{attribute addProperty BoxType "EPP3314-0002-0016"}
{attribute addProperty Id "TC_Inputs_ChannelAT %I*ARRAY[0..6] OF TC_Inputs_Channel_F16A160D128160WcStateAT %I*WcState_98A4DF7520.250InfoDataAT %I*InfoData_BC63D37F80100"}
{attribute addProperty CRC "2970462671"}
{attribute addProperty SizeInBites "210"}
{attribute addProperty SizeInBytes "26.25"}
TYPE EPP3314_A69716D7 :
STRUCT
	{attribute addProperty Name "TC_Inputs_Channel"}
	TC_Inputs_Channel : ARRAY[0..6] OF TC_Inputs_Channel_F16A160D;
	{attribute addProperty Name "WcState"}
	WcState : WcState_98A4DF75;
	{attribute addProperty Name "InfoData"}
	InfoData : InfoData_BC63D37F;
END_STRUCT
END_TYPE

(* stored: Version 1.2.0.0, ProductVersion 3.1.4024.9
   DUT EPP3314_A69716D7: Id {9373b7df-13d8-4dd1-b992-27e49e19af24} *)
